{attribute 'linkalways'} 
{attribute 'no_explicit_call' := 'This FB is a CLASS and must be accessed using methods or properties'}
{attribute 'enable_dynamic_creation'}
FUNCTION_BLOCK Node_F_VN_AdjustSearchWindowOrientationToLinearEdge EXTENDS VisionNode
VAR
	ipSrcImage : _ITcVnImage;
    aStartPoint : _TcVnPoint2_REAL;
    aEndPoint : _TcVnPoint2_REAL;
	eEdgeDirection : _ETcVnEdgeDirection(ETcVnEdgeDirection.TCVN_ED_DARK_TO_LIGHT);
    fMinStrength : _REAL(0.0);
    nMaxThickness : _UDINT(1);
    nSearchLines : _UDINT(1);
    hrPrev : _HRESULT(S_OK);
	hresult : _HRESULT(S_OK);
END_VAR

METHOD PUBLIC  Clone : I_Node
VAR
	pNode : POINTER TO Node_F_VN_AdjustSearchWindowOrientationToLinearEdge;
END_VAR
pNode := __NEW(Node_F_VN_AdjustSearchWindowOrientationToLinearEdge);
Clone := pNode^;
END_METHOD

METHOD FB_init : BOOL
VAR_INPUT
	bInitRetains : BOOL; // if TRUE, the retain variables are initialized (warm start / cold start)
	bInCopyCode : BOOL;  // if TRUE, the instance afterwards gets moved into the copy code (online change)
END_VAR
AddInput('ipSrcImage', ipSrcImage);
AddInput('aStartPoint', aStartPoint);
AddInput('aEndPoint', aEndPoint);
AddParameter('eEdgeDirection', eEdgeDirection);
AddParameter('fMinStrength', fMinStrength);
AddParameter('nMaxThickness', nMaxThickness);
AddParameter('nSearchLines', nSearchLines);
AddInput('hrPrev', hrPrev);
AddOutput('hresult',hresult);
END_METHOD

METHOD PROTECTED OnExecute
hresult.Value := F_VN_AdjustSearchWindowOrientationToLinearEdge(
	ipSrcImage := ipSrcImage.Value,
    aStartPoint := aStartPoint.Value,
    aEndPoint := aEndPoint.Value,
    eEdgeDirection := eEdgeDirection.Value,
	fMinStrength := fMinStrength.Value,
    nMaxThickness := nMaxThickness.Value,
	nSearchLines := nSearchLines.Value,
	hrPrev := hrPrev.Value);
END_METHOD

METHOD PUBLIC PreExecutionCheck
VAR_INPUT
	Check : I_PreExecutionChecks;
END_VAR
Check.IsTrue(ipSrcImage.IsValid, 'ipSrcImage must contain an image');
Check.IsTrue(ipSrcImage.HasChannelCount(1), 'ipSrcImage must contain 1 channel');
Check.IsTrue(nSearchLines.IsOdd, 'nSearchLines must be an odd number');
END_METHOD

END_FUNCTION_BLOCK

(* stored: Version 1.1.0.1, ProductVersion 3.1.4024.13
   POU Node_F_VN_AdjustSearchWindowOrientationToLinearEdge: Id {90501261-b500-4592-9180-d73bee9373a2}, SpecialFunc None
   Folder Constructor: Id {52762dcf-8c4d-4464-9a84-e296006455a1}
   Method Clone: Id {68a5145d-b96f-4b38-8f59-0986d931d1ca}
   Method FB_init: Id {635b2668-e5c8-48d2-adb0-0d457ce15b5d}
   Method OnExecute: Id {50de2c65-fb0e-4bd0-96fa-1ddd811445d3}
   Method PreExecutionCheck: Id {c5dc5531-69b0-45b8-81b7-e06222cb0b91} *)
